SUBAPPLICATION Uebung_039a_sub_Outputs (* Subapplication Type *)
  (* Standard: 61499-2; Description: Copyright (c) 2024 Meisterschulen am Ostbahnhof This program and the accompanying materials are made available under the terms of the Eclipse Public License 2.0 which is available at https://www.eclipse.org/legal/epl-2.0/ SPDX-License-Identifier: EPL-2.0 *)
  (* Version 1.0, 2024-03-03, Franz Höpfinger, Meisterschulen am Ostbahnhof *)
  PACKAGE Uebungen;
  IMPORT SoftKeyActivationCode::SK_RELEASED;
  IMPORT isobus::ut::IDs::ID_NULL;
  IMPORT logiBUS::io::DQ::logiBUS_DO;
  IMPORT logiBUS::io::DQ::logiBUS_DO_S;
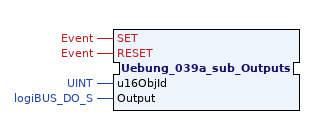
  EVENT_INPUT
    SET; (* Set Output *)
    RESET; (* Reset Output *)
  END_EVENT
  VAR_INPUT
    u16ObjId : UINT := ID_NULL; (* Object ID Softkey/Button *)
    Output : logiBUS::io::DQ::logiBUS_DO_S := logiBUS_DO::Invalid;
  END_VAR
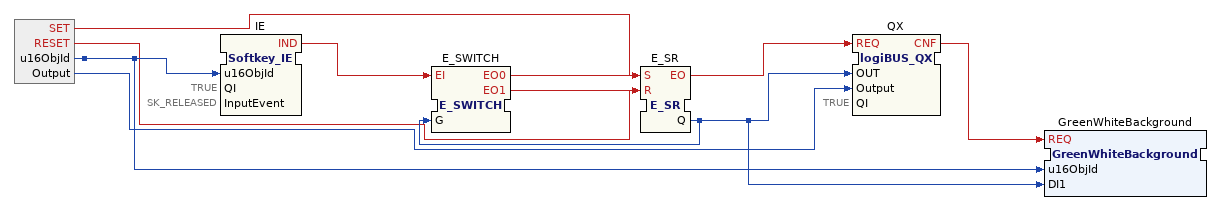
  FBS
    QX : logiBUS::io::DQ::logiBUS_QX(QI := TRUE);
    E_SWITCH : iec61499::events::E_SWITCH;
    E_SR : iec61499::events::E_SR;
    IE : Softkey_IE(QI := TRUE, InputEvent := SK_RELEASED);
  END_FBS
  SUBAPPS
    GreenWhiteBackground : Uebungen::sys::GreenWhiteBackground;
  END_SUBAPPS
  EVENT_CONNECTIONS
    QX.CNF TO GreenWhiteBackground.REQ;
    E_SWITCH.EO0 TO E_SR.S;
    E_SWITCH.EO1 TO E_SR.R;
    IE.IND TO E_SWITCH.EI;
    E_SR.EO TO QX.REQ;
    SET TO E_SR.S;
    RESET TO E_SR.R;
  END_CONNECTIONS
  DATA_CONNECTIONS
    u16ObjId TO GreenWhiteBackground.u16ObjId;
    E_SR.Q TO E_SWITCH.G;
    E_SR.Q TO QX.OUT;
    E_SR.Q TO GreenWhiteBackground.DI1;
    u16ObjId TO IE.u16ObjId;
    Output TO QX.Output;
  END_CONNECTIONS
END_SUBAPPLICATION
